{attribute 'pack_mode' := '1'}
TYPE AxisStatus EXTENDS OutgoingMessage :
STRUCT
	axisIndex: INT; (* 1 or 2. *)
	enabled: BOOL; (* Axis enabled? *)
	moving: BOOL;  (* Axis moving? *)
	atHome: BOOL;   (* Axis has been homed? *)
	atLowLimit: BOOL; (* Axis at low limit switch? *)
	atHighLimit: BOOL; (* Axis at high limit switch? *)
	errorCode: DINT;
	position: LREAL;
END_STRUCT
END_TYPE

(* stored: Version 1.1.0.1, ProductVersion 3.1.4022.12
   DUT AxisStatus: Id {4e2d7ba6-10fa-4462-8ae7-889eed73b54e} *)
